FUNCTION_BLOCK FB_CTManagerWeu EXTENDS FB_CTManager
VAR_INPUT
END_VAR
VAR_OUTPUT
END_VAR
VAR
  fbContainerInstances    : ARRAY[0..lC_MAX_CTS-1] OF FB_ContainerWeu;   // NOTE: 0 based array like base in library
END_VAR

SUPER^();

// call specific CT implementation
nCtr := 0;
WHILE nCtr < nListCount DO
  nIndx := ((nListTail + nCtr) MOD lC_MAX_CTS);    // calculate element index in list
  
  // cyclic call of CT body
  fbContainerInstances[nIndx]();
  
  nCtr := nCtr + 1;
END_WHILE

(*
  Get specific container reference (pointer) from container interface.
*)
METHOD PUBLIC GetContainerInstance : POINTER TO FB_ContainerWeu
VAR_INPUT
  iCT              : I_CT;          (*container at triggered event position*)
END_VAR
VAR
  nCtSel             : UDINT;
END_VAR
IF iCT = 0 THEN LogError(Msg:='GetContainerInstance invalid container'); RETURN; END_IF
nCtSel := iCT.pCT^.nMemIndex;
IF nCtSel < lC_MAX_CTS THEN
  GetContainerInstance := ADR( fbContainerInstances[nCtSel] );
END_IF
END_METHOD

METHOD Init
VAR
  nCtr      : UDINT;
END_VAR
// init FB_CTManager(base) list (interface I_CT) with specific Container instances (FBs) 
FOR nCtr := 0 TO lC_MAX_CTS-1 DO
  iContainerList[nCtr] := fbContainerInstances[nCtr];
END_FOR

// call parent init
SUPER^.InitBase(bAutoDelete := FALSE);
END_METHOD

END_FUNCTION_BLOCK

(* stored: Version 1.1.0.1, ProductVersion 3.1.4024.3
   POU FB_CTManagerWeu: Id {6878a0c6-f16e-440d-ac17-2ecdd0bc47f2}, SpecialFunc None
   Method GetContainerInstance: Id {0f1c4f38-1ca5-4f06-a6b9-0f0cc9dd9309}
   Method Init: Id {80dd4363-7e5b-432c-a24e-3ab3e404e69b} *)
